FUNCTION_BLOCK TestCall IMPLEMENTS I_Callable
VAR_INPUT
END_VAR
VAR_OUTPUT
END_VAR
VAR
	nUdint		: UDINT;
END_VAR

METHOD Call
VAR_INPUT
	iArg	: StageCore.I_Arg;
END_VAR
nUdint := nUdint + 1;
END_METHOD

END_FUNCTION_BLOCK

(* stored: Version 1.1.0.1
   POU TestCall: Id {63bf87f7-0b4f-48aa-9c4a-68cb8ea6de73}, SpecialFunc None
   Method Call: Id {15292887-d3e9-461d-a796-2836f6919931} *)
